Staubli VAL3: _IsUseingBox.pgx

public program _IsUseingBox(bool& x_bNothing[])
  local string l_sEmpty
begin
  x_bNothing=true

  if  first(sml:box)!="" or first(big:box)!=""
    x_bNothing=false
  endIf
end
